TYPE ST_GROUP_CTRL :
STRUCT
  Cmd               : E_GROUP_CTRL;
END_STRUCT
END_TYPE

(* stored: Version 1.1.0.1, ProductVersion 3.1.4024.12
   DUT ST_GROUP_CTRL: Id {5b1697d4-23a2-454c-8797-178dfa194b37} *)
